# EPICS autosave request: iocBoot/iocsri/auto_positions.req
file sri_settings.req P=$(P)
